// TIA Portal V20 export
FUNCTION_BLOCK "FB_Cognex"   // FB55, SCL
{ S7_Optimized_Access := 'TRUE' }
// stored: AutoNumber false, MemoryReserve 100, SetENOAutomatically false
   VAR
      sASTriggerReadyMemo : Bool;
      sASTriggerAckMemo : Bool;
      sASAcquiringMemo : Bool;
      sASMissedTrigMemo : Bool;
      sASOfflineResBit1Memo : Bool;
      sASOfflineResBit2Memo : Bool;
      sASOfflineResBit3Memo : Bool;
      sASOnlineMemo : Bool;
      sISInspectingMemo : Bool;
      sISToggleInspectDoneMemo : Bool;
      sISBufferOverrunMemo : Bool;
      sISResultsValidMemo : Bool;
      sISJobLoadingMemo : Bool;
      sISJobLoadCompleteMemo : Bool;
      sISJobLoadFailedMemo : Bool;
      sISSetUserDataACkMemo : Bool;
      sISJobPassMemo : Bool;
      sSEC0AckMemo : Bool;
      sSEC1AckMemo : Bool;
      sSEC2AckMemo : Bool;
      sSEC3AckMemo : Bool;
      sSEC4AckMemo : Bool;
      sSEC5AckMemo : Bool;
      sSEC6AckMemo : Bool;
      sSEC7AckMemo : Bool;
      sACTriggerEnableMemo : Bool;
      sACTriggerMemo : Bool;
      sACClearAcquirComplMemo : Bool;
      sACSetOfflineMemo : Bool;
      sICBufferResultsEnMemo : Bool;
      sICInspectResultsAckMemo : Bool;
      sICSetUserDataMemo : Bool;
      sICExecuteCmdMemo : Bool;
      sCCSetJobIDMemo : Int;
      sSEC0Memo : Bool;
      sSEC1Memo : Bool;
      sSEC2Memo : Bool;
      sSEC3Memo : Bool;
      sSEC4Memo : Bool;
      sSEC5Memo : Bool;
      sSEC6Memo : Bool;
      sSEC7Memo : Bool;
      sCamLightOn : Bool;
      sUserDataWrite : Bool;
      sUserDataWriteEn : Bool;
      sStartCapture : Bool;
      sAfterResultSoft7 : Bool;
      sTrigAckMemory : Bool;
      sMemoM55 : Bool;
      sSetSetup : Bool;
      sResultDataErrorBit : Bool;
      sICBufferResultsEnPositiveFront : Bool;
      sUserResultReadHole : Bool;
      sUserDataErrorBit : Bool;
      sIRActHoleNrResultMemo : Byte;
      sSetJobId : Int;
      sSetJobIdMemo : Int;
      sJCJobIDMemo : Word;
      sIRInspectionIDMemo : Word;
      sIRInspectResultCodeMemo : Word;
      sASAcquiNumMemo : Word;
      sUserDataErrorCode : Int;
      sResultDataErrorCode : Int;
      sNumChannel : Int;
      sCountAcquiNr : Int;
      sCounter : CTUD_INT;
      sUserDataArray : Array[0..7] of DWord;
      sResultDataArray : Array[0..3] of DWord;
   END_VAR
BEGIN
   REGION Acquisition status
       #sASTriggerReadyMemo := "ASTriggerReady";
       #sASTriggerAckMemo := "ASTriggerAck";
       #sASAcquiringMemo := "ASAcquiring";
       #sASMissedTrigMemo := "ASMissedTrig";
       #sASOfflineResBit1Memo := "ASOfflineResBit1";
       #sASOfflineResBit2Memo := "ASOfflineResBit2";
       #sASOfflineResBit3Memo := "ASOfflineResBit3";
       #sASOnlineMemo := "ASOnline";
       #sASAcquiNumMemo := "ASAcquiNum";
   END_REGION

   REGION Inspection status
       #sISInspectingMemo := "ISInspecting";
       #sISToggleInspectDoneMemo := "ISToggleInspectDone";
       #sISBufferOverrunMemo := "ISBufferOverrun";
       #sISResultsValidMemo := "ISResultsValid";
       #sISJobLoadingMemo := "ISJobLoading";
       "LBP_AlarmMsgs".UserA[8].A70UUxx[41] := "ISJobLoading";
       #sISJobLoadCompleteMemo := "ISJobLoadComplete";
       #sISJobLoadFailedMemo := "ISJobLoadFailed";
       #sISSetUserDataACkMemo := "ISSetUserDataACk";
       #sISJobPassMemo := "ISJobPass";
   END_REGION

   REGION Soft event control output MODule
       #sSEC0AckMemo := "SEC0Ack";
       #sSEC1AckMemo := "SEC1Ack";
       #sSEC2AckMemo := "SEC2Ack";
       #sSEC3AckMemo := "SEC3Ack";
       #sSEC4AckMemo := "SEC4Ack";
       #sSEC5AckMemo := "SEC5Ack";
       #sSEC6AckMemo := "SEC6Ack";
       #sSEC7AckMemo := "SEC7Ack";
   END_REGION

   REGION Job control
       #sJCJobIDMemo := "JCJobID";
   END_REGION

   REGION Inspection result
       #sIRInspectionIDMemo := "IRInspectionID";
       #sIRInspectResultCodeMemo := "IRInspectResultCode";

   END_REGION


   REGION Part programme <-> cognex
       IF #sASOnlineMemo THEN
           // RID if missed trig
           "LBP_AlarmMsgs".ChanA[1].FDD_RID_5C01xx[10] := #sICBufferResultsEnMemo AND #sASMissedTrigMemo;

           // Start camera and set buffer valid
           IF "LBP_Chan1".MDyn[52] THEN    // M52 : Enable buffer and restart the counter hole
               #sICBufferResultsEnMemo := TRUE;
               #sACTriggerEnableMemo := TRUE;
               "LBP_AlarmMsgs".Chan[1].RID[0] := TRUE;
               #sSEC5Memo := FALSE;
           END_IF;

           IF #sASTriggerReadyMemo THEN
               "LBP_AlarmMsgs".Chan[1].RID[0] := FALSE;
           END_IF;

           IF "LBP_Chan1".A_Reset THEN
               #sICBufferResultsEnMemo := FALSE;
               #sACTriggerEnableMemo := FALSE;
               "LBP_AlarmMsgs".Chan[1].RID[0] := FALSE;
               #sSEC5Memo := FALSE;
           END_IF;

           // M53 holes param to Cognex and start capture
           IF "LBP_Chan1".MDyn[53] THEN
               #sUserDataWrite := TRUE;
               #sUserDataWriteEn := TRUE;
               "LBP_AlarmMsgs".Chan[1].RID[11] := TRUE;
           END_IF;

           IF "LBP_Chan1".A_Reset THEN
               #sUserDataWrite := FALSE;
               #sUserDataWriteEn := FALSE;
               "LBP_AlarmMsgs".Chan[1].RID[11] := FALSE;
               #sStartCapture := FALSE;
           END_IF;

           // M54 start acquisition
           IF "LBP_Chan1".MDyn[54] THEN
               #sStartCapture := TRUE;
               "LBP_AlarmMsgs".Chan[1].RID[1] := TRUE;
           END_IF;

           #sACClearAcquirComplMemo :="LBP_Chan1".MDyn[54];

           #sCounter.CU := #sStartCapture AND #sASTriggerReadyMemo AND NOT #sCounter.QU;

           IF #sStartCapture AND #sASTriggerReadyMemo AND NOT #sCounter.QU THEN
               #sACTriggerMemo := TRUE;
               #sAfterResultSoft7 := TRUE;
           END_IF;

           IF #sASTriggerAckMemo THEN
               #sACTriggerMemo := FALSE;
               #sTrigAckMemory := TRUE;
           END_IF;

           IF #sTrigAckMemory AND #sASAcquiringMemo THEN
               #sStartCapture := FALSE;
               "LBP_AlarmMsgs".Chan[1].RID[1] := FALSE;
               #sTrigAckMemory := FALSE;
           END_IF;

           #sCounter.R := "LBP_Chan1".A_Reset;

           IF "LBP_Chan1".A_Reset THEN
               "LBP_AlarmMsgs".Chan[1].RID[1] := FALSE;
               #sACTriggerMemo := FALSE;
           END_IF;

           // M55 end measure
           IF "LBP_Chan1".MDyn[55] AND #sICBufferResultsEnMemo THEN
               "LBP_AlarmMsgs".Chan[1].RID[2] := TRUE;
               #sMemoM55 := TRUE;
               #sSEC6Memo := FALSE;
           END_IF;

           IF (#sMemoM55 AND NOT #sCounter.QU) OR "LBP_Chan1".A_Reset THEN
               #sMemoM55 := FALSE;
               #sACTriggerEnableMemo := FALSE;
               #sSEC5Memo := TRUE;
           END_IF;

           IF #sSEC5AckMemo THEN
               #sSEC5Memo := FALSE;
           END_IF;

               // End part programme <-> cognex
               "LBP_AlarmMsgs".UserA[8].A70UUxx[0] := FALSE;
               "LBP_AlarmMsgs".Chan[1].RID[3] := FALSE;

       ELSE
           IF "LBP_Chan1".MDyn[52]
               OR "LBP_Chan1".MDyn[53]
               OR "LBP_Chan1".MDyn[54]
               OR "LBP_Chan1".MDyn[55] THEN
               "LBP_AlarmMsgs".UserA[8].A70UUxx[0] := TRUE;
               "LBP_AlarmMsgs".Chan[1].RID[3] := TRUE;
           END_IF;

           IF "LBP_Chan1".A_Reset THEN
                "LBP_AlarmMsgs".UserA[8].A70UUxx[0] := FALSE;
                "LBP_AlarmMsgs".Chan[1].RID[3] := FALSE;
           END_IF;

       END_IF;
   END_REGION

   REGION Inspection control
       IF #sISSetUserDataACkMemo AND #sICSetUserDataMemo THEN
           #sICSetUserDataMemo := FALSE;
           #sSEC6Memo := FALSE;
       END_IF;

       IF #sSEC6Memo AND #sSEC6AckMemo THEN
           #sSEC6Memo := FALSE;
           "LBP_AlarmMsgs".Chan[1].RID[11] := FALSE;
       END_IF;
   END_REGION



   REGION Acquisition control
       "ACTriggerEnable" := #sACTriggerEnableMemo;
       "ACTrigger" := #sACTriggerMemo;
       "ACClearAcquirCompl" := #sACClearAcquirComplMemo;
       "ACSetOffline" := #sACSetOfflineMemo;
   END_REGION

   REGION Inspection control
       "ICBufferResultsEn" := #sICBufferResultsEnMemo;
       "ICInspectResultsAck" := #sICInspectResultsAckMemo;
       "ICSetUserData" := #sICSetUserDataMemo;
       "ICExecuteCmd" := #sICExecuteCmdMemo;

       IF #sISSetUserDataACkMemo AND #sICSetUserDataMemo THEN
           #sICSetUserDataMemo := FALSE;
           #sSEC6Memo := TRUE;
       END_IF;

       IF #sSEC6AckMemo AND #sSEC6Memo THEN
           #sSEC6Memo := FALSE;
           "LBP_AlarmMsgs".Chan[1].RID[11] := FALSE;
       END_IF;

   END_REGION

   REGION Job control in setup
       IF "LBP_Chan1".MDyn[58] THEN
           #sSetSetup := TRUE;
           "LBP_AlarmMsgs".Chan[1].RID[13] := TRUE;
       ELSE
           #sSetJobId :=  REAL_TO_INT(ROUND("LBP_Chan1".H1));
       END_IF;

       IF "LBP_Chan1".MDyn[59] THEN
           #sSetSetup := FALSE;
           "LBP_AlarmMsgs".Chan[1].RID[13] := TRUE;
       END_IF;

       IF "LBP_Chan1".A_Reset THEN
           #sSetSetup := FALSE;
           "LBP_AlarmMsgs".Chan[1].RID[13] := FALSE;
           #sICExecuteCmdMemo := FALSE;
           #sACSetOfflineMemo := FALSE;
       END_IF;

   END_REGION

   REGION Job control
       IF #sSetSetup THEN
           // Set new job
           #sSetJobIdMemo := #sSetJobId;
           // If actual job in camera is not the new one AND cmd in progress
           IF NOT (#sSetJobIdMemo = #sJCJobIDMemo
               AND NOT "ICExecuteCmd") THEN
               // Set offline to load job
               IF #sASOnlineMemo THEN
                   #sACSetOfflineMemo := TRUE;
               ELSE
                   // Load job
                   IF NOT #sICExecuteCmdMemo THEN
                       #sCCSetJobIDMemo := #sSetJobIdMemo;
                       #sICExecuteCmdMemo := TRUE;
                   ELSE
                       // Wait job is loaded
                       IF #sISJobLoadCompleteMemo THEN
                           // Reset cmd
                           #sICExecuteCmdMemo := FALSE;
                           #sACSetOfflineMemo := FALSE;
                           "LBP_AlarmMsgs".Chan[1].RID[13] := FALSE;
                           // If load failed
                           IF #sISJobLoadFailedMemo THEN
                               #sICExecuteCmdMemo := FALSE;
                               #sACSetOfflineMemo := FALSE;
                           END_IF;
                       END_IF;
                    END_IF;
               END_IF;
           END_IF;
       END_IF;

   END_REGION

   REGION Soft event control
       "SEC0" := #sSEC0Memo;
       "SEC1" := #sSEC1Memo;
       "SEC2" := #sSEC2Memo;
       "SEC3" := #sSEC3Memo;
       "SEC4" := #sSEC4Memo;
       "SEC5" := #sSEC5Memo;
       "SEC6" := #sSEC6Memo;
       "SEC7" := #sSEC7Memo;

       IF "LBP_Chan1".MDyn[55] OR "LBP_Chan1".A_Reset THEN
           #sSEC0Memo := FALSE;
           #sSEC1Memo := FALSE;
           #sSEC2Memo := FALSE;
           #sSEC3Memo := FALSE;
           #sSEC4Memo := FALSE;
           //#SEC5Memo := FALSE;
           #sSEC6Memo := FALSE;
           #sSEC7Memo := FALSE;
       END_IF;
   END_REGION

   REGION User data from NC
       // If part program send M code
       IF #sUserDataWrite THEN
           // Read data from part program
           "LBP_TransferSelData"(Enable:=#sUserDataWrite,
                                 Funct:=B#16#3,
                                 IVAR1:=8,
                                 IVAR2:=-1,
                                 Error=>#sUserDataErrorBit,
                                 ErrCode=>#sUserDataErrorCode,
                                 S7Var:=#sUserDataArray);

           IF NOT #sUserDataErrorBit THEN
               "UserDataToCognex0" := #sUserDataArray[0];
               "UserDataToCognex1" := #sUserDataArray[1];
               "UserDataToCognex2" := #sUserDataArray[2];
               "UserDataToCognex3" := #sUserDataArray[3];
               "UserDataToCognex4" := #sUserDataArray[4];
               "UserDataToCognex5" := #sUserDataArray[5];
               "UserDataToCognex6" := #sUserDataArray[6];
               "UserDataToCognex7" := #sUserDataArray[7];
           END_IF;

           IF #sUserDataWriteEn AND NOT #sUserDataWrite THEN
               #sUserDataWrite := FALSE;
           END_IF;

           IF #sUserDataWriteEn AND NOT #sUserDataErrorBit THEN
               #sICSetUserDataMemo := FALSE;
               #sUserDataWrite := FALSE;
           END_IF;
       END_IF;

   END_REGION

   REGION Result data to NC
       // Check if cognex has something new
       IF #sISResultsValidMemo AND #sICBufferResultsEnMemo AND NOT #sICBufferResultsEnPositiveFront THEN
           #sUserResultReadHole := TRUE;

           IF #sAfterResultSoft7 THEN
               #sAfterResultSoft7 := FALSE;
               #sSEC4Memo := TRUE;
           END_IF;

           // Define which hole
           IF "IRActHoleNrResult" < 10 THEN
               #sIRActHoleNrResultMemo := "IRActHoleNrResult";
           ELSE
               #sIRActHoleNrResultMemo := 1;
           END_IF;

           #sNumChannel := #sIRActHoleNrResultMemo * 16 + 40;

           // Send result to part program
           #sResultDataArray[0] := "ResultDataFromCognex0";
           #sResultDataArray[1] := "ResultDataFromCognex1";
           #sResultDataArray[2] := "ResultDataFromCognex2";
           #sResultDataArray[3] := "ResultDataFromCognex3";

           "LBP_TransferSelData"(Enable := #sUserResultReadHole,
                                 Funct := B#16#4,
                                 IVAR1 := #sNumChannel,
                                 IVAR2 := -1,
                                 Error => #sResultDataErrorBit,
                                 ErrCode => #sUserDataErrorCode,
                                 S7Var := #sResultDataArray);


       END_IF;

       // Acknowledgements
       #sICBufferResultsEnPositiveFront := #sICBufferResultsEnMemo;

       #sCounter.CD := NOT #sResultDataErrorBit AND #sUserResultReadHole;

       IF NOT #sResultDataErrorBit AND #sUserResultReadHole THEN
           #sUserResultReadHole := FALSE;
           #sICInspectResultsAckMemo := TRUE;

       END_IF;

       #sCountAcquiNr := #sCounter.CV;

       IF NOT #sISResultsValidMemo OR "LBP_Chan1".A_Reset THEN
           #sICInspectResultsAckMemo := FALSE;
       END_IF;

       IF #sSEC4AckMemo THEN
           #sSEC4Memo := FALSE;
       END_IF;

       IF "LBP_Chan1".A_Reset THEN
           #sUserResultReadHole := FALSE;
       END_IF;
   END_REGION
END_FUNCTION_BLOCK
